Universal Robots PolyScope program: Robo22_PakBot_V3_29052022.urp

Program Robo22_PakBot_V3_29052022 (installation=default directory=/programs createdIn=3.15.3.106223 lastSavedIn=3.15.3.106223 robotSerialNumber=2017356754)
Calibrated DH parameters: a=[0.000143, -0.288951, -0.374086, 0.000016, 0.000141, 0]; d=[0.089467, 105.421175, -89.394324, -15.916775, 0.094869, 0.082507]; alpha=[1.569959, -0.002961, -0.007373, 1.570203, -1.570449, 0]; deltaTheta=[0.000042, -0.82396, 0.51794, 0.305959, 0.000026, -0.00009]
Robot Program (runOnlyOnce=false)
  wp_origin := p[0,0,0,0,0,0]
  wp_KeyOrigin := p[0,0,0,0,0,0]
  wp_CornerOrigin := p[0,0,0,0,0,0]
